Fanuc KAREL source: kd00016.KL

-- PROVISIONAL review KL for V1013-1; original PC SHA256 816fa01629eaf00c2b5be78c5464788b6a5cf9c01b3997d8d45be3bbfd27b2d9
-- Incomplete behavior may be omitted. Consult companion uncertainty JSON. Do not deploy.
PROGRAM KD00016
%NOLOCKGROUP
VAR
  I : INTEGER
  J : INTEGER
  B : BOOLEAN
  R : REAL
  S : STRING[80]
BEGIN
  -- UNRESOLVED_PC offsets 5-12; opcodes 9C,23
  -- UNRESOLVED_PC offsets 17-24; opcodes 22,62
  -- UNRESOLVED_PC offsets 29-33; opcodes 7F
END KD00016
